Fanuc KAREL source: compact_preamble.KL

PROGRAM KB00097
%NOLOCKGROUP
VAR
P1 : STRING[80];P2:INTEGER;P3:INTEGER;P4:INTEGER;P5 : STRING[80];P6:INTEGER
BEGIN
P1='A'
P2=1
P3=1
P4=1
P5='A'
P6=1
GET_TSK_INFO(P1,P2,P3,P4,P5,P6)
END KB00097
